(* IEC 61131-3 sources: verifaps-lib/share/PPU.stold (part 5) *)

(* ---- Scenario12_Final.xml_Crane.st ---- *)
FUNCTION_BLOCK Crane
    VAR_OUTPUT  AnalogCranePressure : INT; END_VAR {*Orwxp*}
    VAR_INPUT  CraneDown : BOOL; END_VAR {*Irwxp*}
    VAR_OUTPUT  CraneLower : BOOL; END_VAR {*Orwxp*}
    VAR_INPUT  CraneOnConveyor : BOOL; END_VAR {*Irwxp*}
    VAR_INPUT  CraneOnMagazin : BOOL; END_VAR {*Irwxp*}
    VAR_INPUT  CranePositionStamp : BOOL; END_VAR {*Irwxp*}
    VAR_INPUT  CraneSucked : BOOL; END_VAR {*Irwxp*}
    VAR_OUTPUT  CraneTurnClockwise : BOOL; END_VAR {*Orwxp*}
    VAR_OUTPUT  CraneTurnCounterclockwise : BOOL; END_VAR {*Orwxp*}
    VAR_INPUT  CraneUp : BOOL; END_VAR {*Irwxp*}
    VAR  Duration1 : TIME := TIME#1.0s500.0ms; END_VAR {*Lrwxp*}
    VAR_INPUT  MagazinCapacitiveSensor : BOOL; END_VAR {*Irwxp*}
    VAR_INPUT  MagazinOpticalSensor : BOOL; END_VAR {*Irwxp*}
    VAR_OUTPUT  MagazinVacuumOff : BOOL; END_VAR {*Orwxp*}
    VAR_OUTPUT  MagazinVacuumOn : BOOL; END_VAR {*Orwxp*}
    VAR  SFCInit : BOOL; END_VAR {*Lrwxp*}
    VAR_INPUT  SFCReset : BOOL; END_VAR {*Irwxp*}
    VAR_INPUT  SliderMovedOut : BOOL; END_VAR {*Irwxp*}
    VAR_INPUT  SliderNotMovedOut : BOOL; END_VAR {*Irwxp*}
    VAR_INPUT  StampLowered : BOOL; END_VAR {*Irwxp*}
    VAR_INPUT  StampSliderFilled : BOOL; END_VAR {*Irwxp*}
    VAR_INPUT  StampSliderSensorMovedOut : BOOL; END_VAR {*Irwxp*}
    VAR_INPUT  StartButtonMagazin : BOOL; END_VAR {*Irwxp*}
    VAR_OUTPUT  StartCommandCrane : BOOL; END_VAR {*Orwxp*}
    VAR_INPUT  StartVar : BOOL; END_VAR {*Irwxp*}
    VAR  TimeDelay_Timer : TON; END_VAR {*Lrwxp*}
    VAR  TimeDelay_Timer_Duration : TIME := TIME#50.0ms; END_VAR {*Lrwxp*}
    VAR  TimeDelay_Timer_interconnect : BOOL; END_VAR {*Lrwxp*}
    VAR  Timer1 : TON; END_VAR {*Lrwxp*}
    VAR_INPUT  WorkpieceReady : BOOL; END_VAR {*Irwxp*}
    VAR  _state : Crane_states_t; END_VAR {*Lrwxp*}
    VAR  _transit : BOOL; END_VAR {*Lrwxp*}
    VAR  actualtime1 : TIME; END_VAR {*Lrwxp*}
    VAR  interconnect : BOOL; END_VAR {*Lrwxp*}
    VAR  interconnectCraneStartCommand : BOOL; END_VAR {*Lrwxp*}

    CASE _state OF
        Crane_states_t#Crane_Go_Up:
            _transit := FALSE;
            CraneLower := FALSE;
            IF CraneUp THEN
                _transit := TRUE;
                _state := Crane_states_t#Step3;
            END_IF;

        Crane_states_t#Crane_Go_Up_White:
            _transit := FALSE;
            CraneLower := FALSE;
            IF CraneUp THEN
                _transit := TRUE;
                _state := Crane_states_t#Step3;
            END_IF;

        Crane_states_t#Crane_Init:
            _transit := FALSE;
            CraneLower := TRUE;
            interconnectCraneStartCommand := FALSE;
            AnalogCranePressure := INT#6000;
            IF CraneDown THEN
                _transit := TRUE;
                _state := Crane_states_t#Crane_Init_2;
            END_IF;

        Crane_states_t#Crane_Init_2:
            _transit := FALSE;
            CraneLower := FALSE;
            IF CraneUp THEN
                _transit := TRUE;
                _state := Crane_states_t#Interstep;
            END_IF;

        Crane_states_t#Crane_Lift_At_Stamp:
            _transit := FALSE;
            CraneLower := FALSE;
            IF CraneUp THEN
                _transit := TRUE;
                _state := Crane_states_t#Crane_Turn_Left_From_Stamp;
            END_IF;

        Crane_states_t#Crane_Lift_At_Stamp2:
            _transit := FALSE;
            CraneLower := FALSE;
            IF CraneUp THEN
                _transit := TRUE;
                _state := Crane_states_t#Crane_Turn_Right_From_Stamp;
            END_IF;

        Crane_states_t#Crane_Lift_Conveyor:
            _transit := FALSE;
            CraneLower := FALSE;
            IF TRUE THEN
                _transit := TRUE;
                _state := Crane_states_t#Interstep;
            END_IF;

        Crane_states_t#Crane_Lift_Conveyor2:
            _transit := FALSE;
            CraneLower := FALSE;
            IF TRUE THEN
                _transit := TRUE;
                _state := Crane_states_t#Interstep;
            END_IF;

        Crane_states_t#Crane_Lift_Conveyor_Black:
            _transit := FALSE;
            CraneLower := FALSE;
            IF CraneUp THEN
                _transit := TRUE;
                _state := Crane_states_t#Crane_Turn_Left_Back_To_Stamp;
            END_IF;

        Crane_states_t#Crane_Lift_Magazin:
            _transit := FALSE;
            CraneLower := FALSE;
            IF CraneUp THEN
                _transit := TRUE;
                _state := Crane_states_t#Crane_Turn_Left_NOT_Metallic;
            END_IF;

        Crane_states_t#Crane_Lift_Magazin_Metallic:
            _transit := FALSE;
            CraneLower := FALSE;
            IF CraneUp THEN
                _transit := TRUE;
                _state := Crane_states_t#Crane_Turn_Left_Metallic;
            END_IF;

        Crane_states_t#Crane_Lift_Magazin_White:
            _transit := FALSE;
            CraneLower := FALSE;
            IF CraneUp THEN
                _transit := TRUE;
                _state := Crane_states_t#Crane_Turn_Left_White;
            END_IF;

        Crane_states_t#Crane_Lift_NOT_Metallic_Black:
            _transit := FALSE;
            CraneLower := FALSE;
            IF CraneUp THEN
                _transit := TRUE;
                _state := Crane_states_t#Crane_Turn_Left_NOT_Metallic_Black;
            END_IF;

        Crane_states_t#Crane_Lower:
            _transit := FALSE;
            MagazinVacuumOn := TRUE;
            MagazinVacuumOff := FALSE;
            CraneLower := TRUE;
            AnalogCranePressure := INT#0;
            IF CraneSucked THEN
                _transit := TRUE;
                _state := Crane_states_t#Step0;
            END_IF;

        Crane_states_t#Crane_On_Conveyor:
            _transit := FALSE;
            CraneTurnCounterclockwise := FALSE;
            CraneTurnClockwise := FALSE;
            CraneLower := TRUE;
            IF CraneDown THEN
                _transit := TRUE;
                _state := Crane_states_t#release;
            END_IF;

        Crane_states_t#Crane_On_Conveyor_Metallic:
            _transit := FALSE;
            CraneTurnCounterclockwise := FALSE;
            CraneTurnClockwise := FALSE;
            CraneLower := TRUE;
            IF CraneDown THEN
                _transit := TRUE;
                _state := Crane_states_t#release;
            END_IF;

        Crane_states_t#Crane_On_Conveyor_Metallic2:
            _transit := FALSE;
            CraneTurnCounterclockwise := FALSE;
            CraneTurnClockwise := FALSE;
            CraneLower := TRUE;
            IF CraneDown THEN
                _transit := TRUE;
                _state := Crane_states_t#release2;
            END_IF;

        Crane_states_t#Crane_On_Conveyor_Not_Metallica_Black:
            _transit := FALSE;
            CraneTurnCounterclockwise := FALSE;
            CraneTurnClockwise := FALSE;
            CraneLower := TRUE;
            IF CraneDown THEN
                _transit := TRUE;
                _state := Crane_states_t#release_Black;
            END_IF;

        Crane_states_t#Crane_On_Stamp_Metallic:
            _transit := FALSE;
            CraneTurnCounterclockwise := FALSE;
            CraneTurnClockwise := FALSE;
            CraneLower := TRUE;
            IF CraneDown THEN
                _transit := TRUE;
                _state := Crane_states_t#release_Workpiece;
            END_IF;

        Crane_states_t#Crane_On_Stamp_Metallic2:
            _transit := FALSE;
            CraneTurnCounterclockwise := FALSE;
            CraneTurnClockwise := FALSE;
            IF StampLowered THEN
                _transit := TRUE;
                _state := Crane_states_t#Interstep_4;
            END_IF;

        Crane_states_t#Crane_On_Stamp_Metallic2_Lower:
            _transit := FALSE;
            CraneLower := TRUE;
            IF CraneDown THEN
                _transit := TRUE;
                _state := Crane_states_t#Suck_At_Stamp2;
            END_IF;

        Crane_states_t#Crane_On_Stamp_Stop_Black:
            _transit := FALSE;
            CraneTurnClockwise := FALSE;
            CraneTurnCounterclockwise := FALSE;
            IF TRUE THEN
                _transit := TRUE;
                _state := Crane_states_t#Reset_interconnect;
            END_IF;

        Crane_states_t#Crane_On_Stamp_White:
            _transit := FALSE;
            CraneTurnCounterclockwise := FALSE;
            CraneTurnClockwise := FALSE;
            CraneLower := TRUE;
            IF CraneDown THEN
                _transit := TRUE;
                _state := Crane_states_t#release_Workpiece_White;
            END_IF;

        Crane_states_t#Crane_Turn_Left_Back_To_Stamp:
            _transit := FALSE;
            CraneTurnCounterclockwise := TRUE;
            CraneTurnClockwise := FALSE;
            IF CranePositionStamp THEN
                _transit := TRUE;
                _state := Crane_states_t#Crane_On_Stamp_Stop_Black;
            END_IF;

        Crane_states_t#Crane_Turn_Left_From_Stamp:
            _transit := FALSE;
            CraneTurnClockwise := TRUE;
            CraneTurnCounterclockwise := FALSE;
            IF CraneOnConveyor THEN
                _transit := TRUE;
                _state := Crane_states_t#Crane_On_Conveyor_Metallic;
            END_IF;

        Crane_states_t#Crane_Turn_Left_Metallic:
            _transit := FALSE;
            CraneTurnCounterclockwise := TRUE;
            CraneTurnClockwise := FALSE;
            IF CranePositionStamp THEN
                _transit := TRUE;
                _state := Crane_states_t#Crane_On_Stamp_Metallic;
            END_IF;

        Crane_states_t#Crane_Turn_Left_Metallic2:
            _transit := FALSE;
            CraneTurnCounterclockwise := TRUE;
            CraneTurnClockwise := FALSE;
            IF CranePositionStamp THEN
                _transit := TRUE;
                _state := Crane_states_t#Crane_On_Stamp_Metallic2;
            END_IF;

        Crane_states_t#Crane_Turn_Left_NOT_Metallic:
            _transit := FALSE;
            CraneTurnCounterclockwise := TRUE;
            CraneTurnClockwise := FALSE;
            IF CraneOnConveyor THEN
                _transit := TRUE;
                _state := Crane_states_t#Crane_On_Conveyor;
            END_IF;

        Crane_states_t#Crane_Turn_Left_NOT_Metallic_Black:
            _transit := FALSE;
            CraneTurnCounterclockwise := TRUE;
            CraneTurnClockwise := FALSE;
            IF CraneOnConveyor THEN
                _transit := TRUE;
                _state := Crane_states_t#Crane_On_Conveyor_Not_Metallica_Black;
            END_IF;

        Crane_states_t#Crane_Turn_Left_White:
            _transit := FALSE;
            CraneTurnCounterclockwise := TRUE;
            CraneTurnClockwise := FALSE;
            IF CranePositionStamp THEN
                _transit := TRUE;
                _state := Crane_states_t#Crane_On_Stamp_White;
            END_IF;

        Crane_states_t#Crane_Turn_Right_From_Stamp:
            _transit := FALSE;
            CraneTurnClockwise := TRUE;
            CraneTurnCounterclockwise := FALSE;
            IF CraneOnConveyor THEN
                _transit := TRUE;
                _state := Crane_states_t#Crane_On_Conveyor_Metallic2;
            END_IF;

        Crane_states_t#Init:
            _transit := FALSE;
            IF TRUE THEN
                _transit := TRUE;
                _state := Crane_states_t#Start_Crane;
            END_IF;

        Crane_states_t#Interstep:
            _transit := FALSE;
            StartCommandCrane := TRUE;
            IF StartVar THEN
                _transit := TRUE;
                _state := Crane_states_t#Interstep_2;
            END_IF;

        Crane_states_t#Interstep_2:
            _transit := FALSE;
            IF SliderMovedOut THEN
                _transit := TRUE;
                _state := Crane_states_t#TimeDelay;
            END_IF;

        Crane_states_t#Interstep_3:
            _transit := FALSE;
            IF NOT WorkpieceReady THEN
                _transit := TRUE;
                _state := Crane_states_t#No_Workpiece_ready;
            ELSEIF WorkpieceReady THEN
                _transit := TRUE;
                _state := Crane_states_t#Turn_Right;
            END_IF;

        Crane_states_t#Interstep_4:
            _transit := FALSE;
            IF StampSliderSensorMovedOut THEN
                _transit := TRUE;
                _state := Crane_states_t#Crane_On_Stamp_Metallic2_Lower;
            END_IF;

        Crane_states_t#Lower_Crane:
            _transit := FALSE;
            CraneLower := TRUE;
            IF CraneDown THEN
                _transit := TRUE;
                _state := Crane_states_t#Suck_At_Stamp;
            END_IF;

        Crane_states_t#Magazin_Stop:
            _transit := FALSE;
            CraneTurnClockwise := FALSE;
            CraneTurnCounterclockwise := FALSE;
            IF TRUE THEN
                _transit := TRUE;
                _state := Crane_states_t#Crane_Lower;
            END_IF;

        Crane_states_t#Magazin_Stop_Black:
            _transit := FALSE;
            CraneTurnClockwise := FALSE;
            CraneTurnCounterclockwise := FALSE;
            MagazinVacuumOn := TRUE;
            MagazinVacuumOff := FALSE;
            CraneLower := TRUE;
            IF CraneSucked THEN
                _transit := TRUE;
                _state := Crane_states_t#Crane_Lift_NOT_Metallic_Black;
            END_IF;

        Crane_states_t#Magazin_Stop_Final:
            _transit := FALSE;
            CraneTurnClockwise := FALSE;
            CraneTurnCounterclockwise := FALSE;
            IF TRUE THEN
                _transit := TRUE;
                _state := Crane_states_t#Start_Crane;
            END_IF;

        Crane_states_t#No_Workpiece_ready:
            _transit := FALSE;
            MagazinVacuumOn := FALSE;
            MagazinVacuumOff := FALSE;
            CraneLower := FALSE;
            IF StampSliderFilled THEN
                _transit := TRUE;
                _state := Crane_states_t#Crane_Turn_Left_Metallic2;
            ELSEIF NOT StampSliderFilled THEN
                _transit := TRUE;
                _state := Crane_states_t#Turn_Right_Final;
            END_IF;

        Crane_states_t#Reset_interconnect:
            _transit := FALSE;
            interconnect := FALSE;
            Timer1(IN := FALSE, PT := TIME#1.0ms);
            IF SliderMovedOut THEN
                _transit := TRUE;
                _state := Crane_states_t#Lower_Crane;
            END_IF;

        Crane_states_t#Stamp_Pressure_Profile_Set_Metallic:
            _transit := FALSE;
            AnalogCranePressure := INT#7000;
            IF TRUE THEN
                _transit := TRUE;
                _state := Crane_states_t#Crane_Lift_Magazin_Metallic;
            END_IF;

        Crane_states_t#Stamp_Pressure_Profile_Set_White:
            _transit := FALSE;
            AnalogCranePressure := INT#6000;
            IF TRUE THEN
                _transit := TRUE;
                _state := Crane_states_t#Crane_Lift_Magazin_White;
            END_IF;

        Crane_states_t#Start_Crane:
            _transit := FALSE;
            CraneLower := FALSE;
            MagazinVacuumOff := FALSE;
            MagazinVacuumOn := FALSE;
            CraneTurnCounterclockwise := FALSE;
            CraneTurnClockwise := FALSE;
            AnalogCranePressure := INT#0;
            StartVar := FALSE;
            StartCommandCrane := FALSE;
            IF (StartButtonMagazin = TRUE) THEN
                interconnectCraneStartCommand := TRUE;
            END_IF;
            IF interconnectCraneStartCommand THEN
                _transit := TRUE;
                _state := Crane_states_t#Crane_Init;
            END_IF;

        Crane_states_t#Step0:
            _transit := FALSE;
            IF (NOT MagazinCapacitiveSensor AND MagazinOpticalSensor) THEN
                _transit := TRUE;
                _state := Crane_states_t#Stamp_Pressure_Profile_Set_White;
            ELSEIF (MagazinCapacitiveSensor AND MagazinOpticalSensor) THEN
                _transit := TRUE;
                _state := Crane_states_t#Stamp_Pressure_Profile_Set_Metallic;
            ELSEIF (NOT MagazinCapacitiveSensor AND NOT MagazinOpticalSensor) THEN
                _transit := TRUE;
                _state := Crane_states_t#Crane_Lift_Magazin;
            END_IF;

        Crane_states_t#Step2:
            _transit := FALSE;
            IF (NOT MagazinCapacitiveSensor AND NOT MagazinOpticalSensor) THEN
                _transit := TRUE;
                _state := Crane_states_t#Turn_Right_Black;
            ELSEIF (MagazinCapacitiveSensor OR MagazinOpticalSensor) THEN
                _transit := TRUE;
                _state := Crane_states_t#pause;
            END_IF;

        Crane_states_t#Step3:
            _transit := FALSE;
            IF NOT WorkpieceReady THEN
                _transit := TRUE;
                _state := Crane_states_t#Step4;
            ELSEIF WorkpieceReady THEN
                _transit := TRUE;
                _state := Crane_states_t#Step2;
            END_IF;

        Crane_states_t#Step4:
            _transit := FALSE;
            IF TRUE THEN
                _transit := TRUE;
                _state := Crane_states_t#Interstep;
            END_IF;

        Crane_states_t#Suck_At_Stamp:
            _transit := FALSE;
            MagazinVacuumOn := TRUE;
            MagazinVacuumOff := FALSE;
            IF CraneSucked THEN
                _transit := TRUE;
                _state := Crane_states_t#Crane_Lift_At_Stamp;
            END_IF;

        Crane_states_t#Suck_At_Stamp2:
            _transit := FALSE;
            MagazinVacuumOn := TRUE;
            MagazinVacuumOff := FALSE;
            IF CraneSucked THEN
                _transit := TRUE;
                _state := Crane_states_t#Crane_Lift_At_Stamp2;
            END_IF;

        Crane_states_t#TimeDelay:
            _transit := FALSE;
            TimeDelay_Timer(IN := TRUE, PT := TimeDelay_Timer_Duration);
            TimeDelay_Timer_interconnect := TimeDelay_Timer.Q;
            IF TimeDelay_Timer_interconnect THEN
                _transit := TRUE;
                _state := Crane_states_t#Interstep_3;
            END_IF;

        Crane_states_t#Turn_Right:
            _transit := FALSE;
            CraneTurnClockwise := TRUE;
            CraneTurnCounterclockwise := FALSE;
            IF CraneOnMagazin THEN
                _transit := TRUE;
                _state := Crane_states_t#Magazin_Stop;
            END_IF;

        Crane_states_t#Turn_Right_Black:
            _transit := FALSE;
            CraneTurnClockwise := TRUE;
            CraneTurnCounterclockwise := FALSE;
            IF CraneOnMagazin THEN
                _transit := TRUE;
                _state := Crane_states_t#Magazin_Stop_Black;
            END_IF;

        Crane_states_t#Turn_Right_Final:
            _transit := FALSE;
            CraneTurnClockwise := TRUE;
            CraneTurnCounterclockwise := FALSE;
            AnalogCranePressure := INT#0;
            IF CraneOnMagazin THEN
                _transit := TRUE;
                _state := Crane_states_t#Magazin_Stop_Final;
            END_IF;

        Crane_states_t#pause:
            _transit := FALSE;
            Timer1(IN := CraneUp, PT := Duration1);
            interconnect := Timer1.Q;
            IF interconnect THEN
                _transit := TRUE;
                _state := Crane_states_t#Reset_interconnect;
            END_IF;

        Crane_states_t#release:
            _transit := FALSE;
            MagazinVacuumOff := TRUE;
            MagazinVacuumOn := FALSE;
            IF TRUE THEN
                _transit := TRUE;
                _state := Crane_states_t#Crane_Lift_Conveyor;
            END_IF;

        Crane_states_t#release2:
            _transit := FALSE;
            MagazinVacuumOff := TRUE;
            MagazinVacuumOn := FALSE;
            IF TRUE THEN
                _transit := TRUE;
                _state := Crane_states_t#Crane_Lift_Conveyor2;
            END_IF;

        Crane_states_t#release_Black:
            _transit := FALSE;
            MagazinVacuumOn := FALSE;
            MagazinVacuumOff := TRUE;
            IF TRUE THEN
                _transit := TRUE;
                _state := Crane_states_t#Crane_Lift_Conveyor_Black;
            END_IF;

        Crane_states_t#release_Workpiece:
            _transit := FALSE;
            MagazinVacuumOff := TRUE;
            MagazinVacuumOn := FALSE;
            IF TRUE THEN
                _transit := TRUE;
                _state := Crane_states_t#Crane_Go_Up;
            END_IF;

        Crane_states_t#release_Workpiece_White:
            _transit := FALSE;
            MagazinVacuumOff := TRUE;
            MagazinVacuumOn := FALSE;
            IF TRUE THEN
                _transit := TRUE;
                _state := Crane_states_t#Crane_Go_Up_White;
            END_IF;

            END_CASE;
END_FUNCTION_BLOCK

(* ---- Scenario12_Final.xml_Magazin.st ---- *)
FUNCTION_BLOCK Magazin
    VAR_INPUT  CraneDown : BOOL; END_VAR {*Irwxp*}
    VAR_OUTPUT  CraneLower : BOOL; END_VAR {*Orwxp*}
    VAR_INPUT  CraneOnConveyor : BOOL; END_VAR {*Irwxp*}
    VAR_INPUT  CraneOnMagazin : BOOL; END_VAR {*Irwxp*}
    VAR_INPUT  CraneSucked : BOOL; END_VAR {*Irwxp*}
    VAR_OUTPUT  CraneTurnClockwise : BOOL; END_VAR {*Orwxp*}
    VAR_OUTPUT  CraneTurnCounterclockwise : BOOL; END_VAR {*Orwxp*}
    VAR_INPUT  CraneUp : BOOL; END_VAR {*Irwxp*}
    VAR_OUTPUT  MagazinGreenLamp : BOOL; END_VAR {*Orwxp*}
    VAR_OUTPUT  MagazinSlider : BOOL; END_VAR {*Orwxp*}
    VAR_OUTPUT  MagazinVacuumOff : BOOL; END_VAR {*Orwxp*}
    VAR_OUTPUT  MagazinVacuumOn : BOOL; END_VAR {*Orwxp*}
    VAR_OUTPUT  MagazinWhiteLamp : BOOL; END_VAR {*Orwxp*}
    VAR  SFCInit : BOOL; END_VAR {*Lrwxp*}
    VAR_INPUT  SFCReset : BOOL; END_VAR {*Irwxp*}
    VAR_INPUT  SliderMovedOut : BOOL; END_VAR {*Irwxp*}
    VAR_INPUT  SliderNotMovedOut : BOOL; END_VAR {*Irwxp*}
    VAR_INPUT  StartButtonMagazin : BOOL; END_VAR {*Irwxp*}
    VAR_OUTPUT  StartCommandMagazin : BOOL; END_VAR {*Orwxp*}
    VAR_INPUT  StartVar : BOOL; END_VAR {*Irwxp*}
    VAR_INPUT  WorkpieceReady : BOOL; END_VAR {*Irwxp*}
    VAR  _state : Magazin_states_t; END_VAR {*Lrwxp*}
    VAR  _transit : BOOL; END_VAR {*Lrwxp*}
    VAR  interconnectMagazinStartCommand : BOOL; END_VAR {*Lrwxp*}

    CASE _state OF
        Magazin_states_t#Green_Lamp:
            _transit := FALSE;
            MagazinGreenLamp := TRUE;
            interconnectMagazinStartCommand := FALSE;
            IF TRUE THEN
                _transit := TRUE;
                _state := Magazin_states_t#Magazin_Init;
            END_IF;

        Magazin_states_t#Init:
            _transit := FALSE;
            IF TRUE THEN
                _transit := TRUE;
                _state := Magazin_states_t#Start_Magazin;
            END_IF;

        Magazin_states_t#Interstep:
            _transit := FALSE;
            StartCommandMagazin := TRUE;
            IF StartVar THEN
                _transit := TRUE;
                _state := Magazin_states_t#convey;
            END_IF;

        Magazin_states_t#Magazin_Init:
            _transit := FALSE;
            MagazinSlider := TRUE;
            IF TRUE THEN
                _transit := TRUE;
                _state := Magazin_states_t#Magazin_Init_2;
            END_IF;

        Magazin_states_t#Magazin_Init_2:
            _transit := FALSE;
            MagazinSlider := FALSE;
            IF TRUE THEN
                _transit := TRUE;
                _state := Magazin_states_t#Interstep;
            END_IF;

        Magazin_states_t#Slider_Move_Back:
            _transit := FALSE;
            IF ((SliderMovedOut = TRUE) AND (SliderNotMovedOut = FALSE)) THEN
                MagazinSlider := FALSE;
            END_IF;
            IF CraneUp THEN
                _transit := TRUE;
                _state := Magazin_states_t#Step1;
            END_IF;

        Magazin_states_t#Start_Magazin:
            _transit := FALSE;
            MagazinSlider := FALSE;
            MagazinGreenLamp := FALSE;
            StartVar := FALSE;
            StartCommandMagazin := FALSE;
            IF (StartButtonMagazin = TRUE) THEN
                interconnectMagazinStartCommand := TRUE;
            END_IF;
            IF interconnectMagazinStartCommand THEN
                _transit := TRUE;
                _state := Magazin_states_t#Green_Lamp;
            END_IF;

        Magazin_states_t#Step0:
            _transit := FALSE;
            IF CraneDown THEN
                _transit := TRUE;
                _state := Magazin_states_t#Slider_Move_Back;
            END_IF;

        Magazin_states_t#Step1:
            _transit := FALSE;
            IF CraneOnConveyor THEN
                _transit := TRUE;
                _state := Magazin_states_t#Interstep;
            END_IF;

        Magazin_states_t#convey:
            _transit := FALSE;
            IF SliderNotMovedOut THEN
                MagazinSlider := TRUE;
            END_IF;
            IF CraneOnMagazin THEN
                _transit := TRUE;
                _state := Magazin_states_t#Step0;
            END_IF;

            END_CASE;
END_FUNCTION_BLOCK

(* ---- Scenario12_Final.xml_Pusher.st ---- *)
FUNCTION_BLOCK Pusher
    VAR  Duration2 : TIME := TIME#2.0s; END_VAR {*Lrwxp*}
    VAR  Duration3 : TIME := TIME#200.0ms; END_VAR {*Lrwxp*}
    VAR  Duration_Slide1_Black : TIME := TIME#900.0ms; END_VAR {*Lrwxp*}
    VAR  Duration_Slide1_Metal : TIME := TIME#320.0ms; END_VAR {*Lrwxp*}
    VAR  Duration_Slide1_White : TIME := TIME#320.0ms; END_VAR {*Lrwxp*}
    VAR  Duration_Slide2_Black : TIME := TIME#2.0s; END_VAR {*Lrwxp*}
    VAR  Duration_Slide2_Metal : TIME := TIME#390.0ms; END_VAR {*Lrwxp*}
    VAR  Duration_Slide2_White : TIME := TIME#390.0ms; END_VAR {*Lrwxp*}
    VAR  Priority_Var_Black : INT := INT#3; END_VAR {*Lrwxp*}
    VAR  Priority_Var_Metal : INT := INT#3; END_VAR {*Lrwxp*}
    VAR  Priority_Var_White : INT := INT#3; END_VAR {*Lrwxp*}
    VAR_OUTPUT  PusherY1 : BOOL; END_VAR {*Orwxp*}
    VAR_OUTPUT  PusherY2 : BOOL; END_VAR {*Orwxp*}
    VAR  SFCInit : BOOL; END_VAR {*Lrwxp*}
    VAR_INPUT  SFCReset : BOOL; END_VAR {*Irwxp*}
    VAR  Slide1_black : INT := INT#1; END_VAR {*Lrwxp*}
    VAR  Slide1_metal : INT := INT#1; END_VAR {*Lrwxp*}
    VAR  Slide1_white : INT := INT#1; END_VAR {*Lrwxp*}
    VAR  Slide2_black : INT := INT#1; END_VAR {*Lrwxp*}
    VAR  Slide2_metal : INT := INT#1; END_VAR {*Lrwxp*}
    VAR  Slide2_white : INT := INT#1; END_VAR {*Lrwxp*}
    VAR  Slide3_black : INT := INT#1; END_VAR {*Lrwxp*}
    VAR  Slide3_metal : INT := INT#1; END_VAR {*Lrwxp*}
    VAR  Slide3_white : INT := INT#1; END_VAR {*Lrwxp*}
    VAR_INPUT  SorterCapacitiveSensorPusher1 : BOOL; END_VAR {*Irwxp*}
    VAR_INPUT  SorterCapacitiveSensorPusher2 : BOOL; END_VAR {*Irwxp*}
    VAR_INPUT  SorterLightbarrierCraneInterface : BOOL; END_VAR {*Irwxp*}
    VAR_INPUT  SorterLightnessSensorPusher1 : BOOL; END_VAR {*Irwxp*}
    VAR_INPUT  SorterLightnessSensorPusher2 : BOOL; END_VAR {*Irwxp*}
    VAR_INPUT  SorterLightnessSensorPusher3 : BOOL; END_VAR {*Irwxp*}
    VAR_INPUT  SorterLightnesssensorCraneInterfaceInverse : BOOL; END_VAR {*Irwxp*}
    VAR_INPUT  SorterPusher1MovedIn : BOOL; END_VAR {*Irwxp*}
    VAR_INPUT  SorterPusher1MovedOut : BOOL; END_VAR {*Irwxp*}
    VAR_INPUT  SorterPusher2MovedIn : BOOL; END_VAR {*Irwxp*}
    VAR_INPUT  SorterPusher2MovedOut : BOOL; END_VAR {*Irwxp*}
    VAR_INPUT  SorterStartButton : BOOL; END_VAR {*Irwxp*}
    VAR_INPUT  StartVar : BOOL; END_VAR {*Irwxp*}
    VAR  Timer2 : TON; END_VAR {*Lrwxp*}
    VAR  Timer3 : TON; END_VAR {*Lrwxp*}
    VAR  Timer_Slide1_Black : TON; END_VAR {*Lrwxp*}
    VAR  Timer_Slide1_Metal : TON; END_VAR {*Lrwxp*}
    VAR  Timer_Slide1_White : TON; END_VAR {*Lrwxp*}
    VAR  Timer_Slide2_Black : TON; END_VAR {*Lrwxp*}
    VAR  Timer_Slide2_Metal : TON; END_VAR {*Lrwxp*}
    VAR  Timer_Slide2_White : TON; END_VAR {*Lrwxp*}
    VAR  _state : Pusher_states_t; END_VAR {*Lrwxp*}
    VAR  _transit : BOOL; END_VAR {*Lrwxp*}
    VAR  interconnect2 : BOOL; END_VAR {*Lrwxp*}
    VAR  interconnect3 : BOOL; END_VAR {*Lrwxp*}
    VAR  interconnect_Slide1_Black : BOOL; END_VAR {*Lrwxp*}
    VAR  interconnect_Slide1_Metal : BOOL; END_VAR {*Lrwxp*}
    VAR  interconnect_Slide1_White : BOOL; END_VAR {*Lrwxp*}
    VAR  interconnect_Slide2_Black : BOOL; END_VAR {*Lrwxp*}
    VAR  interconnect_Slide2_Metal : BOOL; END_VAR {*Lrwxp*}
    VAR  interconnect_Slide2_White : BOOL; END_VAR {*Lrwxp*}

    CASE _state OF
        Pusher_states_t#Check_For_Black:
            _transit := FALSE;
            IF ((Slide3_black = INT#1) AND (Priority_Var_Black = INT#3)) THEN
                _transit := TRUE;
                _state := Pusher_states_t#Third_Slide_black_workpieces;
            ELSEIF ((Slide2_black = INT#1) AND (Priority_Var_Black = INT#2)) THEN
                _transit := TRUE;
                _state := Pusher_states_t#Second_Slide_black_workpieces;
            ELSEIF ((Slide1_black = INT#1) AND (Priority_Var_Black = INT#1)) THEN
                _transit := TRUE;
                _state := Pusher_states_t#First_Slide_black_workpieces;
            END_IF;

        Pusher_states_t#Check_For_Metal:
            _transit := FALSE;
            IF ((Slide3_metal = INT#1) AND (Priority_Var_Metal = INT#3)) THEN
                _transit := TRUE;
                _state := Pusher_states_t#Third_Slide_metal_workpieces;
            ELSEIF ((Slide2_metal = INT#1) AND (Priority_Var_Metal = INT#2)) THEN
                _transit := TRUE;
                _state := Pusher_states_t#Second_Slide_metal_workpieces;
            ELSEIF ((Slide1_metal = INT#1) AND (Priority_Var_Metal = INT#1)) THEN
                _transit := TRUE;
                _state := Pusher_states_t#First_Slide_metal_workpieces;
            END_IF;

        Pusher_states_t#Check_For_White:
            _transit := FALSE;
            IF ((Slide1_white = INT#1) AND (Priority_Var_White = INT#1)) THEN
                _transit := TRUE;
                _state := Pusher_states_t#First_Slide_white_workpieces;
            ELSEIF ((Slide2_white = INT#1) AND (Priority_Var_White = INT#2)) THEN
                _transit := TRUE;
                _state := Pusher_states_t#Second_Slide_white_workpieces;
            ELSEIF ((Slide3_white = INT#1) AND (Priority_Var_White = INT#3)) THEN
                _transit := TRUE;
                _state := Pusher_states_t#Third_Slide_white_workpieces;
            END_IF;

        Pusher_states_t#First_Slide_Timer_Black:
            _transit := FALSE;
            IF (SorterLightnesssensorCraneInterfaceInverse = TRUE) THEN
                Timer_Slide1_Black(IN := SorterLightnesssensorCraneInterfaceInverse, PT := Duration_Slide1_Black);
                interconnect_Slide1_Black := Timer_Slide1_Black.Q;
            END_IF;
            IF interconnect_Slide1_Black THEN
                _transit := TRUE;
                _state := Pusher_states_t#PusherY1_Move_Out_Black;
            END_IF;

        Pusher_states_t#First_Slide_Timer_Metal:
            _transit := FALSE;
            Timer_Slide1_Metal(IN := TRUE, PT := Duration_Slide1_Metal);
            interconnect_Slide1_Metal := Timer_Slide1_Metal.Q;
            IF interconnect_Slide1_Metal THEN
                _transit := TRUE;
                _state := Pusher_states_t#PusherY1_Move_Out_Metal;
            END_IF;

        Pusher_states_t#First_Slide_Timer_White:
            _transit := FALSE;
            Timer_Slide1_White(IN := TRUE, PT := Duration_Slide1_White);
            interconnect_Slide1_White := Timer_Slide1_White.Q;
            IF interconnect_Slide1_White THEN
                _transit := TRUE;
                _state := Pusher_states_t#PusherY1_Move_Out_White;
            END_IF;

        Pusher_states_t#First_Slide_black_workpieces:
            _transit := FALSE;
            IF TRUE THEN
                _transit := TRUE;
                _state := Pusher_states_t#First_Slide_Timer_Black;
            END_IF;

        Pusher_states_t#First_Slide_metal_workpieces:
            _transit := FALSE;
            IF TRUE THEN
                _transit := TRUE;
                _state := Pusher_states_t#First_Slide_Timer_Metal;
            END_IF;

        Pusher_states_t#First_Slide_white_workpieces:
            _transit := FALSE;
            IF TRUE THEN
                _transit := TRUE;
                _state := Pusher_states_t#First_Slide_Timer_White;
            END_IF;

        Pusher_states_t#Init:
            _transit := FALSE;
            IF StartVar THEN
                _transit := TRUE;
                _state := Pusher_states_t#Interstep;
            END_IF;

        Pusher_states_t#Interstep:
            _transit := FALSE;
            PusherY1 := FALSE;
            PusherY2 := FALSE;
            interconnect2 := FALSE;
            interconnect3 := FALSE;
            StartVar := FALSE;
            interconnect_Slide1_Black := FALSE;
            interconnect_Slide2_Black := FALSE;
            interconnect_Slide1_White := FALSE;
            interconnect_Slide2_White := FALSE;
            interconnect_Slide1_Metal := FALSE;
            interconnect_Slide2_Metal := FALSE;
            IF TRUE THEN
                _transit := TRUE;
                _state := Pusher_states_t#Interstep_2;
            END_IF;

        Pusher_states_t#Interstep_2:
            _transit := FALSE;
            IF ((SorterLightnessSensorPusher1 AND NOT SorterCapacitiveSensorPusher1) AND (Priority_Var_White > INT#0)) THEN
                _transit := TRUE;
                _state := Pusher_states_t#Check_For_White;
            ELSEIF ((SorterLightnessSensorPusher1 AND SorterCapacitiveSensorPusher1) AND (Priority_Var_Metal > INT#0)) THEN
                _transit := TRUE;
                _state := Pusher_states_t#Check_For_Metal;
            ELSEIF ((NOT SorterLightnesssensorCraneInterfaceInverse AND SorterLightbarrierCraneInterface) AND (Priority_Var_Black > INT#0)) THEN
                _transit := TRUE;
                _state := Pusher_states_t#Check_For_Black;
            END_IF;

        Pusher_states_t#PusherY1_Move_In_Black:
            _transit := FALSE;
            IF ((SorterPusher1MovedOut = TRUE) AND (SorterPusher1MovedIn = FALSE)) THEN
                PusherY1 := FALSE;
            END_IF;
            IF SorterPusher1MovedIn THEN
                _transit := TRUE;
                _state := Pusher_states_t#Reset_interconnect_Slide1_Black;
            END_IF;

        Pusher_states_t#PusherY1_Move_In_Metal:
            _transit := FALSE;
            IF ((SorterPusher1MovedOut = TRUE) AND (SorterPusher1MovedIn = FALSE)) THEN
                PusherY1 := FALSE;
            END_IF;
            IF SorterPusher1MovedIn THEN
                _transit := TRUE;
                _state := Pusher_states_t#Reset_interconnect_Slide1_Metal;
            END_IF;

        Pusher_states_t#PusherY1_Move_In_White:
            _transit := FALSE;
            IF ((SorterPusher1MovedOut = TRUE) AND (SorterPusher1MovedIn = FALSE)) THEN
                PusherY1 := FALSE;
            END_IF;
            IF SorterPusher1MovedIn THEN
                _transit := TRUE;
                _state := Pusher_states_t#Reset_interconnect_Slide1_White;
            END_IF;

        Pusher_states_t#PusherY1_Move_Out_Black:
            _transit := FALSE;
            IF ((SorterPusher1MovedOut = FALSE) AND (SorterPusher1MovedIn = TRUE)) THEN
                PusherY1 := TRUE;
            END_IF;
            IF SorterPusher1MovedOut THEN
                _transit := TRUE;
                _state := Pusher_states_t#Wait_Y1_Black;
            END_IF;

        Pusher_states_t#PusherY1_Move_Out_Metal:
            _transit := FALSE;
            IF ((SorterPusher1MovedOut = FALSE) AND (SorterPusher1MovedIn = TRUE)) THEN
                PusherY1 := TRUE;
            END_IF;
            IF SorterPusher1MovedOut THEN
                _transit := TRUE;
                _state := Pusher_states_t#Wait_Y1_Metal;
            END_IF;

        Pusher_states_t#PusherY1_Move_Out_White:
            _transit := FALSE;
            IF ((SorterPusher1MovedOut = FALSE) AND (SorterPusher1MovedIn = TRUE)) THEN
                PusherY1 := TRUE;
            END_IF;
            IF SorterPusher1MovedOut THEN
                _transit := TRUE;
                _state := Pusher_states_t#Wait_Y1_White;
            END_IF;

        Pusher_states_t#PusherY2_Move_In_Black:
            _transit := FALSE;
            IF ((SorterPusher2MovedOut = TRUE) AND (SorterPusher2MovedIn = FALSE)) THEN
                PusherY2 := FALSE;
            END_IF;
            IF SorterPusher2MovedIn THEN
                _transit := TRUE;
                _state := Pusher_states_t#Reset_interconnect_Slide2_Black;
            END_IF;

        Pusher_states_t#PusherY2_Move_In_Metal:
            _transit := FALSE;
            IF ((SorterPusher2MovedOut = TRUE) AND (SorterPusher2MovedIn = FALSE)) THEN
                PusherY2 := FALSE;
            END_IF;
            IF SorterPusher2MovedIn THEN
                _transit := TRUE;
                _state := Pusher_states_t#Reset_interconnect_Slide2_Metal;
            END_IF;

        Pusher_states_t#PusherY2_Move_In_White:
            _transit := FALSE;
            IF ((SorterPusher2MovedOut = TRUE) AND (SorterPusher2MovedIn = FALSE)) THEN
                PusherY2 := FALSE;
            END_IF;
            IF SorterPusher2MovedIn THEN
                _transit := TRUE;
                _state := Pusher_states_t#Reset_interconnect_Slide2_White;
            END_IF;

        Pusher_states_t#PusherY2_Move_Out_Black:
            _transit := FALSE;
            IF ((SorterPusher2MovedOut = FALSE) AND (SorterPusher2MovedIn = TRUE)) THEN
                PusherY2 := TRUE;
            END_IF;
            IF SorterPusher2MovedOut THEN
                _transit := TRUE;
                _state := Pusher_states_t#Wait_Y2_Black;
            END_IF;

        Pusher_states_t#PusherY2_Move_Out_Metal:
            _transit := FALSE;
            IF ((SorterPusher2MovedOut = FALSE) AND (SorterPusher2MovedIn = TRUE)) THEN
                PusherY2 := TRUE;
            END_IF;
            IF SorterPusher2MovedOut THEN
                _transit := TRUE;
                _state := Pusher_states_t#Wait_Y2_Metal;
            END_IF;

        Pusher_states_t#PusherY2_Move_Out_White:
            _transit := FALSE;
            IF ((SorterPusher2MovedOut = FALSE) AND (SorterPusher2MovedIn = TRUE)) THEN
                PusherY2 := TRUE;
            END_IF;
            IF SorterPusher2MovedOut THEN
                _transit := TRUE;
                _state := Pusher_states_t#Wait_Y2_White;
            END_IF;

        Pusher_states_t#Reset_interconnect3:
            _transit := FALSE;
            interconnect3 := FALSE;
            Timer3(IN := FALSE, PT := TIME#);
            Slide3_black := (Slide3_black - INT#1);
            Priority_Var_Black := (Priority_Var_Black - INT#1);
            IF TRUE THEN
                _transit := TRUE;
                _state := Pusher_states_t#Interstep_2;
            END_IF;

        Pusher_states_t#Reset_interconnect_Slide1_Black:
            _transit := FALSE;
            interconnect3 := FALSE;
            Timer3(IN := FALSE, PT := TIME#);
            interconnect_Slide1_Black := FALSE;
            Timer_Slide1_Black(IN := FALSE, PT := TIME#);
            Slide1_black := (Slide1_black - INT#1);
            Priority_Var_Black := (Priority_Var_Black - INT#1);
            IF TRUE THEN
                _transit := TRUE;
                _state := Pusher_states_t#Interstep_2;
            END_IF;

        Pusher_states_t#Reset_interconnect_Slide1_Metal:
            _transit := FALSE;
            interconnect3 := FALSE;
            Timer3(IN := FALSE, PT := TIME#);
            interconnect_Slide1_Metal := FALSE;
            Timer_Slide1_Metal(IN := FALSE, PT := TIME#);
            Slide1_metal := (Slide1_metal - INT#1);
            Priority_Var_Metal := (Priority_Var_Metal - INT#1);
            IF TRUE THEN
                _transit := TRUE;
                _state := Pusher_states_t#Interstep_2;
            END_IF;

        Pusher_states_t#Reset_interconnect_Slide1_White:
            _transit := FALSE;
            interconnect3 := FALSE;
            Timer3(IN := FALSE, PT := TIME#);
            interconnect_Slide1_White := FALSE;
            Timer_Slide1_White(IN := FALSE, PT := TIME#);
            Slide1_white := (Slide1_white - INT#1);
            Priority_Var_White := (Priority_Var_White - INT#1);
            IF TRUE THEN
                _transit := TRUE;
                _state := Pusher_states_t#Interstep_2;
            END_IF;

        Pusher_states_t#Reset_interconnect_Slide2_Black:
            _transit := FALSE;
            interconnect3 := FALSE;
            Timer3(IN := FALSE, PT := TIME#);
            interconnect_Slide2_Black := FALSE;
            Timer_Slide2_Black(IN := FALSE, PT := TIME#);
            Slide2_black := (Slide2_black - INT#1);
            Priority_Var_Black := (Priority_Var_Black - INT#1);
            IF TRUE THEN
                _transit := TRUE;
                _state := Pusher_states_t#Interstep_2;
            END_IF;

        Pusher_states_t#Reset_interconnect_Slide2_Metal:
            _transit := FALSE;
            interconnect3 := FALSE;
            Timer3(IN := FALSE, PT := TIME#);
            interconnect_Slide2_Metal := FALSE;
            Timer_Slide2_Metal(IN := FALSE, PT := TIME#);
            Slide2_metal := (Slide2_metal - INT#1);
            Priority_Var_Metal := (Priority_Var_Metal - INT#1);
            IF TRUE THEN
                _transit := TRUE;
                _state := Pusher_states_t#Interstep_2;
            END_IF;

        Pusher_states_t#Reset_interconnect_Slide2_White:
            _transit := FALSE;
            interconnect3 := FALSE;
            Timer3(IN := FALSE, PT := TIME#);
            interconnect_Slide2_White := FALSE;
            Timer_Slide2_White(IN := FALSE, PT := TIME#);
            Slide2_white := (Slide2_white - INT#1);
            Priority_Var_White := (Priority_Var_White - INT#1);
            IF TRUE THEN
                _transit := TRUE;
                _state := Pusher_states_t#Interstep_2;
            END_IF;

        Pusher_states_t#Reset_interconnect_Slide3_Metal:
            _transit := FALSE;
            interconnect3 := FALSE;
            Timer3(IN := FALSE, PT := TIME#);
            Slide3_metal := (Slide3_metal - INT#1);
            Priority_Var_Metal := (Priority_Var_Metal - INT#1);
            IF TRUE THEN
                _transit := TRUE;
                _state := Pusher_states_t#Interstep_2;
            END_IF;

        Pusher_states_t#Reset_interconnect_Slide3_White:
            _transit := FALSE;
            interconnect3 := FALSE;
            Timer3(IN := FALSE, PT := TIME#);
            Slide3_white := (Slide3_white - INT#1);
            Priority_Var_White := (Priority_Var_White - INT#1);
            IF TRUE THEN
                _transit := TRUE;
                _state := Pusher_states_t#Interstep_2;
            END_IF;

        Pusher_states_t#Second_Slide_Timer_Black:
            _transit := FALSE;
            IF (SorterLightnesssensorCraneInterfaceInverse = TRUE) THEN
                Timer_Slide2_Black(IN := SorterLightnesssensorCraneInterfaceInverse, PT := Duration_Slide2_Black);
                interconnect_Slide2_Black := Timer_Slide2_Black.Q;
            END_IF;
            IF interconnect_Slide2_Black THEN
                _transit := TRUE;
                _state := Pusher_states_t#PusherY2_Move_Out_Black;
            END_IF;

        Pusher_states_t#Second_Slide_Timer_Metal:
            _transit := FALSE;
            Timer_Slide2_Metal(IN := TRUE, PT := Duration_Slide2_Metal);
            interconnect_Slide2_Metal := Timer_Slide2_Metal.Q;
            IF interconnect_Slide2_Metal THEN
                _transit := TRUE;
                _state := Pusher_states_t#PusherY2_Move_Out_Metal;
            END_IF;

        Pusher_states_t#Second_Slide_Timer_White:
            _transit := FALSE;
            Timer_Slide2_White(IN := TRUE, PT := Duration_Slide2_White);
            interconnect_Slide2_White := Timer_Slide2_White.Q;
            IF interconnect_Slide2_White THEN
                _transit := TRUE;
                _state := Pusher_states_t#PusherY2_Move_Out_White;
            END_IF;

        Pusher_states_t#Second_Slide_black_workpieces:
            _transit := FALSE;
            IF TRUE THEN
                _transit := TRUE;
                _state := Pusher_states_t#Second_Slide_Timer_Black;
            END_IF;

        Pusher_states_t#Second_Slide_metal_workpieces:
            _transit := FALSE;
            IF (SorterLightnessSensorPusher2 AND SorterCapacitiveSensorPusher2) THEN
                _transit := TRUE;
                _state := Pusher_states_t#Second_Test_For_Metal;
            END_IF;

        Pusher_states_t#Second_Slide_white_workpieces:
            _transit := FALSE;
            IF (SorterLightnessSensorPusher2 AND NOT SorterCapacitiveSensorPusher2) THEN
                _transit := TRUE;
                _state := Pusher_states_t#Second_Test_For_White;
            END_IF;

        Pusher_states_t#Second_Test_For_Metal:
            _transit := FALSE;
            IF TRUE THEN
                _transit := TRUE;
                _state := Pusher_states_t#Second_Slide_Timer_Metal;
            END_IF;

        Pusher_states_t#Second_Test_For_White:
            _transit := FALSE;
            IF TRUE THEN
                _transit := TRUE;
                _state := Pusher_states_t#Second_Slide_Timer_White;
            END_IF;

        Pusher_states_t#Third_Slide_black_workpieces:
            _transit := FALSE;
            IF (NOT SorterLightnessSensorPusher2 AND NOT SorterCapacitiveSensorPusher2) THEN
                _transit := TRUE;
                _state := Pusher_states_t#Wait_Black;
            END_IF;

        Pusher_states_t#Third_Slide_metal_workpieces:
            _transit := FALSE;
            IF (SorterLightnessSensorPusher2 AND SorterCapacitiveSensorPusher2) THEN
                _transit := TRUE;
                _state := Pusher_states_t#Wait_Metal;
            END_IF;

        Pusher_states_t#Third_Slide_white_workpieces:
            _transit := FALSE;
            IF (SorterLightnessSensorPusher2 AND NOT SorterCapacitiveSensorPusher2) THEN
                _transit := TRUE;
                _state := Pusher_states_t#Wait_White;
            END_IF;

        Pusher_states_t#Wait_Black:
            _transit := FALSE;
            IF ((NOT SorterLightnessSensorPusher2 AND NOT SorterCapacitiveSensorPusher2) = TRUE) THEN
                Timer2(IN := (NOT SorterLightnessSensorPusher2 AND NOT SorterCapacitiveSensorPusher2), PT := Duration2);
                interconnect2 := Timer2.Q;
            END_IF;
            IF interconnect2 THEN
                _transit := TRUE;
                _state := Pusher_states_t#Reset_interconnect3;
            END_IF;

        Pusher_states_t#Wait_Metal:
            _transit := FALSE;
            Timer3(IN := TRUE, PT := Duration3);
            interconnect3 := Timer3.Q;
            IF interconnect3 THEN
                _transit := TRUE;
                _state := Pusher_states_t#Reset_interconnect_Slide3_Metal;
            END_IF;

        Pusher_states_t#Wait_White:
            _transit := FALSE;
            Timer3(IN := TRUE, PT := Duration3);
            interconnect3 := Timer3.Q;
            IF interconnect3 THEN
                _transit := TRUE;
                _state := Pusher_states_t#Reset_interconnect_Slide3_White;
            END_IF;

        Pusher_states_t#Wait_Y1_Black:
            _transit := FALSE;
            IF (PusherY1 = TRUE) THEN
                Timer3(IN := PusherY1, PT := Duration3);
                interconnect3 := Timer3.Q;
            END_IF;
            IF interconnect3 THEN
                _transit := TRUE;
                _state := Pusher_states_t#PusherY1_Move_In_Black;
            END_IF;

        Pusher_states_t#Wait_Y1_Metal:
            _transit := FALSE;
            IF (PusherY1 = TRUE) THEN
                Timer3(IN := PusherY1, PT := Duration3);
                interconnect3 := Timer3.Q;
            END_IF;
            IF interconnect3 THEN
                _transit := TRUE;
                _state := Pusher_states_t#PusherY1_Move_In_Metal;
            END_IF;

        Pusher_states_t#Wait_Y1_White:
            _transit := FALSE;
            IF (PusherY1 = TRUE) THEN
                Timer3(IN := PusherY1, PT := Duration3);
                interconnect3 := Timer3.Q;
            END_IF;
            IF interconnect3 THEN
                _transit := TRUE;
                _state := Pusher_states_t#PusherY1_Move_In_White;
            END_IF;

        Pusher_states_t#Wait_Y2_Black:
            _transit := FALSE;
            IF (PusherY2 = TRUE) THEN
                Timer3(IN := PusherY2, PT := Duration3);
                interconnect3 := Timer3.Q;
            END_IF;
            IF interconnect3 THEN
                _transit := TRUE;
                _state := Pusher_states_t#PusherY2_Move_In_Black;
            END_IF;

        Pusher_states_t#Wait_Y2_Metal:
            _transit := FALSE;
            IF (PusherY2 = TRUE) THEN
                Timer3(IN := PusherY2, PT := Duration3);
                interconnect3 := Timer3.Q;
            END_IF;
            IF interconnect3 THEN
                _transit := TRUE;
                _state := Pusher_states_t#PusherY2_Move_In_Metal;
            END_IF;

        Pusher_states_t#Wait_Y2_White:
            _transit := FALSE;
            IF (PusherY2 = TRUE) THEN
                Timer3(IN := PusherY2, PT := Duration3);
                interconnect3 := Timer3.Q;
            END_IF;
            IF interconnect3 THEN
                _transit := TRUE;
                _state := Pusher_states_t#PusherY2_Move_In_White;
            END_IF;

            END_CASE;
END_FUNCTION_BLOCK

(* ---- Scenario12_Final.xml_Stamp.st ---- *)
FUNCTION_BLOCK Stamp
    VAR_INPUT  CraneDown : BOOL; END_VAR {*Irwxp*}
    VAR_INPUT  CraneOnConveyor : BOOL; END_VAR {*Irwxp*}
    VAR_INPUT  CranePositionStamp : BOOL; END_VAR {*Irwxp*}
    VAR_INPUT  CraneSucked : BOOL; END_VAR {*Irwxp*}
    VAR_INPUT  CraneUp : BOOL; END_VAR {*Irwxp*}
    VAR  Duration : TIME := TIME#500.0ms; END_VAR {*Lrwxp*}
    VAR  SFCInit : BOOL; END_VAR {*Lrwxp*}
    VAR_INPUT  SFCReset : BOOL; END_VAR {*Irwxp*}
    VAR_OUTPUT  StampGreenLamp : BOOL; END_VAR {*Orwxp*}
    VAR_INPUT  StampLowered : BOOL; END_VAR {*Irwxp*}
    VAR_OUTPUT  StampPressure : BOOL; END_VAR {*Orwxp*}
    VAR_OUTPUT  StampPusher : BOOL; END_VAR {*Orwxp*}
    VAR_INPUT  StampSliderFilled : BOOL; END_VAR {*Irwxp*}
    VAR_OUTPUT  StampSliderMovedIn : BOOL; END_VAR {*Orwxp*}
    VAR_OUTPUT  StampSliderMovedOut : BOOL; END_VAR {*Orwxp*}
    VAR_INPUT  StampSliderSensorMovedIn : BOOL; END_VAR {*Irwxp*}
    VAR_INPUT  StampSliderSensorMovedOut : BOOL; END_VAR {*Irwxp*}
    VAR_INPUT  StampStartButton : BOOL; END_VAR {*Irwxp*}
    VAR_INPUT  StampUp : BOOL; END_VAR {*Irwxp*}
    VAR_OUTPUT  StampWhiteLamp : BOOL; END_VAR {*Orwxp*}
    VAR_OUTPUT  StartCommandStamp : BOOL; END_VAR {*Orwxp*}
    VAR_INPUT  StartVar : BOOL; END_VAR {*Irwxp*}
    VAR  Timer : TON; END_VAR {*Lrwxp*}
    VAR  _state : Stamp_states_t; END_VAR {*Lrwxp*}
    VAR  _transit : BOOL; END_VAR {*Lrwxp*}
    VAR  interconnect : BOOL; END_VAR {*Lrwxp*}
    VAR  interconnectStampStartCommand : BOOL; END_VAR {*Lrwxp*}

    CASE _state OF
        Stamp_states_t#Green_Lamp:
            _transit := FALSE;
            StampGreenLamp := TRUE;
            interconnectStampStartCommand := FALSE;
            IF TRUE THEN
                _transit := TRUE;
                _state := Stamp_states_t#Stamp_Init_1;
            END_IF;

        Stamp_states_t#Init:
            _transit := FALSE;
            IF TRUE THEN
                _transit := TRUE;
                _state := Stamp_states_t#Start_Stamp;
            END_IF;

        Stamp_states_t#Interstep:
            _transit := FALSE;
            StartCommandStamp := TRUE;
            IF StartVar THEN
                _transit := TRUE;
                _state := Stamp_states_t#Intertsep_2;
            END_IF;

        Stamp_states_t#Intertsep_2:
            _transit := FALSE;
            IF StampSliderFilled THEN
                _transit := TRUE;
                _state := Stamp_states_t#Step0;
            END_IF;

        Stamp_states_t#StampProcess:
            _transit := FALSE;
            StampSliderMovedIn := FALSE;
            StampPusher := TRUE;
            IF StampLowered THEN
                _transit := TRUE;
                _state := Stamp_states_t#Step1;
            END_IF;

        Stamp_states_t#StampSliderBack:
            _transit := FALSE;
            StampSliderMovedIn := TRUE;
            StampSliderMovedOut := FALSE;
            IF StampSliderSensorMovedIn THEN
                _transit := TRUE;
                _state := Stamp_states_t#StampProcess;
            END_IF;

        Stamp_states_t#StampSliderForward:
            _transit := FALSE;
            StampPusher := FALSE;
            StampSliderMovedOut := TRUE;
            IF ((StampLowered = FALSE) AND (StampUp = TRUE)) THEN
                interconnect := FALSE;
            END_IF;
            Timer(IN := FALSE, PT := TIME#1.0ms);
            IF StampSliderMovedOut THEN
                _transit := TRUE;
                _state := Stamp_states_t#Step2;
            END_IF;

        Stamp_states_t#Stamp_Init_1:
            _transit := FALSE;
            StampSliderMovedIn := TRUE;
            StampSliderMovedOut := FALSE;
            IF StampSliderSensorMovedIn THEN
                _transit := TRUE;
                _state := Stamp_states_t#Stamp_Init_2;
            END_IF;

        Stamp_states_t#Stamp_Init_2:
            _transit := FALSE;
            StampSliderMovedIn := FALSE;
            StampSliderMovedOut := TRUE;
            IF StampSliderSensorMovedOut THEN
                _transit := TRUE;
                _state := Stamp_states_t#Stamp_Init_3;
            END_IF;

        Stamp_states_t#Stamp_Init_3:
            _transit := FALSE;
            StampPusher := TRUE;
            IF StampLowered THEN
                _transit := TRUE;
                _state := Stamp_states_t#Stamp_Init_4;
            END_IF;

        Stamp_states_t#Stamp_Init_4:
            _transit := FALSE;
            StampPusher := FALSE;
            IF StampUp THEN
                _transit := TRUE;
                _state := Stamp_states_t#Interstep;
            END_IF;

        Stamp_states_t#Start_Stamp:
            _transit := FALSE;
            StampSliderMovedOut := FALSE;
            StampSliderMovedIn := FALSE;
            StampPusher := FALSE;
            StampGreenLamp := FALSE;
            StampPressure := FALSE;
            StartCommandStamp := FALSE;
            IF (StampStartButton = TRUE) THEN
                interconnectStampStartCommand := TRUE;
            END_IF;
            IF interconnectStampStartCommand THEN
                _transit := TRUE;
                _state := Stamp_states_t#Green_Lamp;
            END_IF;

        Stamp_states_t#Step0:
            _transit := FALSE;
            IF CraneUp THEN
                _transit := TRUE;
                _state := Stamp_states_t#StampSliderBack;
            END_IF;

        Stamp_states_t#Step1:
            _transit := FALSE;
            Timer(IN := StampLowered, PT := TIME#);
            interconnect := Timer.Q;
            IF interconnect THEN
                _transit := TRUE;
                _state := Stamp_states_t#StampSliderForward;
            END_IF;

        Stamp_states_t#Step2:
            _transit := FALSE;
            IF (CraneOnConveyor AND NOT StampSliderFilled) THEN
                _transit := TRUE;
                _state := Stamp_states_t#Interstep;
            END_IF;

            END_CASE;
END_FUNCTION_BLOCK
